(* CODESYS project Johnson,Joachim,Uppgift17_V2.project

Project tree, tasks and I/O mapping:
  Device : CODESYS Control Win V3, 3S - Smart Software Solutions GmbH, order no. 305021, version 3.5.10.40
    application Application
      libraries: Standard, * (System)
      task MainTask (cyclic, interval t#20ms, priority 1) calls PLC_PRG, Light [Handling Lights], ResetAlarm, PrintoutErrorMessages
      program PLC_PRG [LD]
      Symbols
      global variables GVL
      program Light [CFC]
      program ResetAlarm [CFC]
      program PrintoutErrorMessages [ST]
*)

// Device/Application/GVL
{attribute 'qualified_only'}
VAR_GLOBAL
		// signals from buttons
	iSUB00_S1: BOOL; // StartButton
	iSUB00_S2: BOOL; // Stopbutton
	iSUB00_S3: BOOL; // Resetbutton
	
	running: BOOL; 	 // Is the aplication running
	alarm: BOOL; 	 // Is the aplication running
	alarmcode: WORD; // handling the codes of the alarm
	
	Alarm1: BOOL;
	Alarm2: BOOL;
	Alarm3: BOOL;
	
	// Signals from conveyors
	iSUB01_B1: BOOL; // Signals för conveyor 1. ontop
	iSUB02_B1: BOOL; // Signals för conveyor 2. ontop
	iSUB03_B1: BOOL; // Signals för conveyor 3. ontop
	
	// Conveyor signal ontop conveyro
	oSUB00_H1: BOOL; // Auto-On light
	oSUB00_H2: BOOL; // Alarm light
	oSUB00_H3: WORD; // Display of errors
	oSUB01_K1: BOOL; // MOTOR FÖR converoyr 1
	oSUB02_K1: BOOL; // MOTOR FÖR converoyr 2
	oSUB03_K1: BOOL; // MOTOR FÖR converoyr 3
END_VAR

// Device/Application/PLC_PRG
PROGRAM PLC_PRG
VAR
	ReturnRunnongBool: BOOL;
	PressBtnTime: TIME;
	PressBtnTimer: TON;
	ONTOPCONRETURN: BOOL;
	ONTOPCONRETURN2: BOOL; // check that the previous con not take controll over engine/converour
	ONTOPCONRETURN3: BOOL; // check that the previous con not take controll over engine/converour
	TON_0: TON;
	TON_1: TON;
	TimElapseSincePastFirstSens: TIME;
	TON_2: TON;
	running: BOOL;
	ErrorCodePrintout: CTD;
	ErrorCodePrintout2: CTD;
	ErrorCodePrintout3: CTD;
	TimElapseSincePastFirstSens2: TIME;
	TON_3: TON;
	TON_4: TON;
	TimElapseSincePastFirstSens3: TIME;
	TimElapseSincePastFirstSens4: TIME;
	Alarm2: BOOL;
	Alarm1: BOOL;
	Alarm3: BOOL;
END_VAR
VAR // added by the converter: edge detectors and wires of the graphical bodies
    _w1, _w2, _w3, _w4, _w5, _w6 : BOOL;
END_VAR

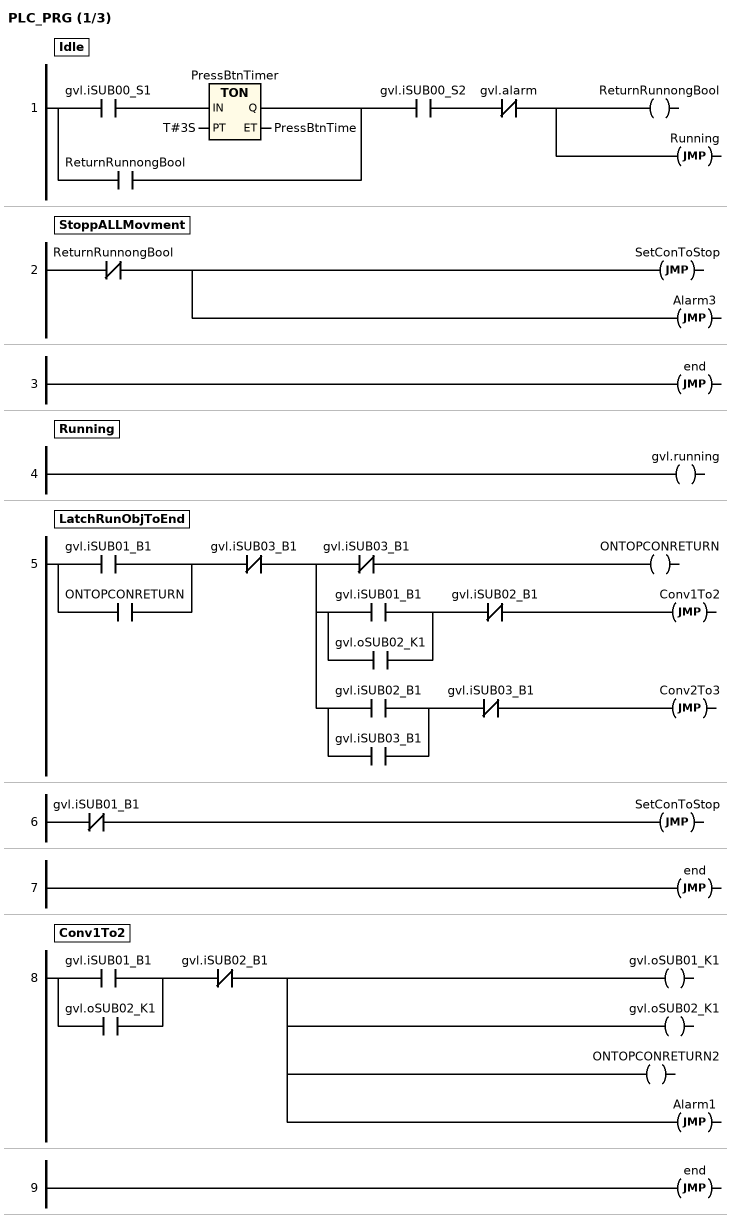
// NETWORK 1
Idle:
PressBtnTimer(IN := gvl.iSUB00_S1, PT := T#3S, ET => PressBtnTime); // TON
_w1 := ((PressBtnTimer.Q OR ReturnRunnongBool) AND gvl.iSUB00_S2) AND NOT gvl.alarm;
ReturnRunnongBool := _w1;
IF _w1 THEN JMP Running; END_IF

// NETWORK 2
StoppALLMovment:
_w2 := NOT ReturnRunnongBool;
IF _w2 THEN JMP SetConToStop; END_IF
IF _w2 THEN JMP Alarm3; END_IF

// NETWORK 3
JMP end;

// NETWORK 4
Running:
gvl.running := TRUE;

// NETWORK 5
LatchRunObjToEnd:
_w3 := (gvl.iSUB01_B1 OR ONTOPCONRETURN) AND NOT gvl.iSUB03_B1;
ONTOPCONRETURN := _w3 AND NOT gvl.iSUB03_B1;
IF (_w3 AND (gvl.iSUB01_B1 OR gvl.oSUB02_K1)) AND NOT gvl.iSUB02_B1 THEN JMP Conv1To2; END_IF
IF _w3 AND (gvl.iSUB02_B1 OR gvl.iSUB03_B1) AND NOT gvl.iSUB03_B1 THEN JMP Conv2To3; END_IF

// NETWORK 6
IF NOT gvl.iSUB01_B1 THEN JMP SetConToStop; END_IF

// NETWORK 7
JMP end;

// NETWORK 8
Conv1To2:
_w4 := (gvl.iSUB01_B1 OR gvl.oSUB02_K1) AND NOT gvl.iSUB02_B1;
gvl.oSUB01_K1 := _w4;
gvl.oSUB02_K1 := _w4;
ONTOPCONRETURN2 := _w4;
IF _w4 THEN JMP Alarm1; END_IF

// NETWORK 9
JMP end;

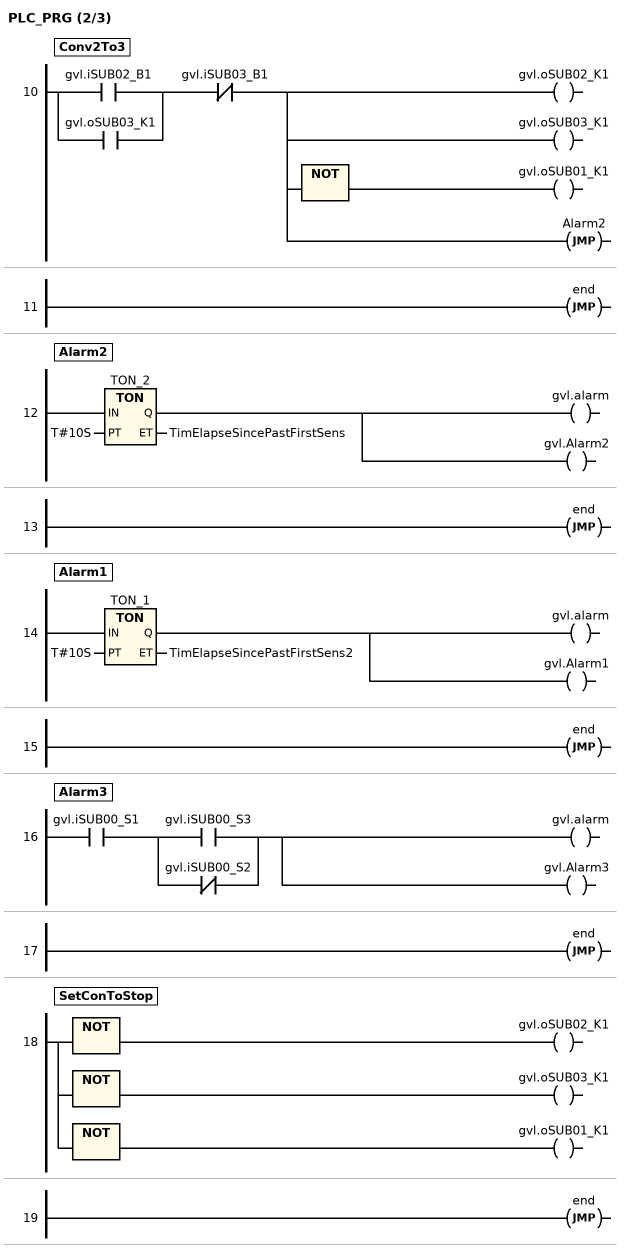
// NETWORK 10
Conv2To3:
_w5 := (gvl.iSUB02_B1 OR gvl.oSUB03_K1) AND NOT gvl.iSUB03_B1;
gvl.oSUB02_K1 := _w5;
gvl.oSUB03_K1 := _w5;
gvl.oSUB01_K1 := NOT _w5;
IF _w5 THEN JMP Alarm2; END_IF

// NETWORK 11
JMP end;

// NETWORK 12
Alarm2:
TON_2(IN := TRUE, PT := T#10S, ET => TimElapseSincePastFirstSens); // TON
gvl.alarm := TON_2.Q;
gvl.Alarm2 := TON_2.Q;

// NETWORK 13
JMP end;

// NETWORK 14
Alarm1:
TON_1(IN := TRUE, PT := T#10S, ET => TimElapseSincePastFirstSens2); // TON
gvl.alarm := TON_1.Q;
gvl.Alarm1 := TON_1.Q;

// NETWORK 15
JMP end;

// NETWORK 16
Alarm3:
_w6 := gvl.iSUB00_S1 AND (gvl.iSUB00_S3 OR NOT gvl.iSUB00_S2);
gvl.alarm := _w6;
gvl.Alarm3 := _w6;

// NETWORK 17
JMP end;

// NETWORK 18
SetConToStop:
gvl.oSUB02_K1 := NOT TRUE;
gvl.oSUB03_K1 := NOT TRUE;
gvl.oSUB01_K1 := NOT TRUE;

// NETWORK 19
JMP end;

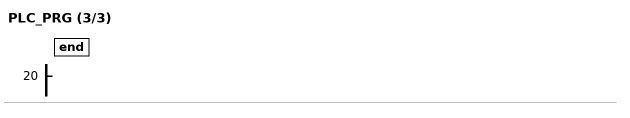
// NETWORK 20
end: ;

END_PROGRAM

// Device/Application/Light
PROGRAM Light
VAR
	Light_Time_TurnOff_Delayf: TON;
	TurnLightOffTimeoutpu: TIME;
	TurnLightOnTimeoutpu: TIME;
	Button_O: TON;
END_VAR
VAR // added by the converter: edge detectors and wires of the graphical bodies
    _w1 : BOOL;
END_VAR

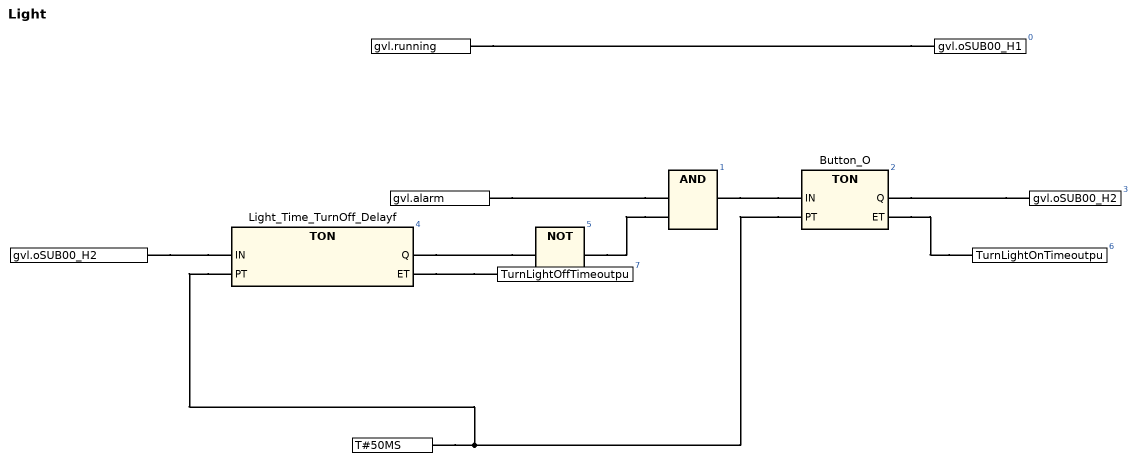
gvl.oSUB00_H1 := gvl.running;
Button_O(IN := gvl.alarm AND _w1, PT := T#50MS); // TON
gvl.oSUB00_H2 := Button_O.Q;
Light_Time_TurnOff_Delayf(IN := gvl.oSUB00_H2, PT := T#50MS); // TON
_w1 := NOT Light_Time_TurnOff_Delayf.Q;
TurnLightOnTimeoutpu := Button_O.ET;
TurnLightOffTimeoutpu := Light_Time_TurnOff_Delayf.ET;

END_PROGRAM

// Device/Application/ResetAlarm
PROGRAM ResetAlarm
VAR
END_VAR
VAR // added by the converter: edge detectors and wires of the graphical bodies
    _w1 : BOOL;
END_VAR

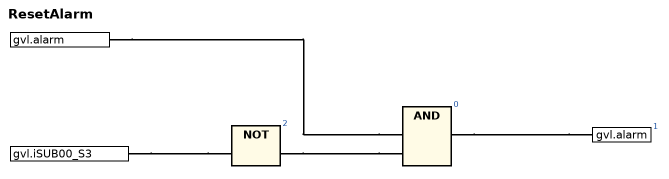
gvl.alarm := gvl.alarm AND _w1;
_w1 := NOT gvl.iSUB00_S3;

END_PROGRAM

// Device/Application/PrintoutErrorMessages
PROGRAM PrintoutErrorMessages
VAR
END_VAR

IF gvl.Alarm1 THEN
	gvl.oSUB00_H3 := 10;
END_IF

IF gvl.Alarm2 THEN
	gvl.oSUB00_H3 := 20;
END_IF

IF gvl.Alarm3 THEN
	gvl.oSUB00_H3 := 30;
END_IF

END_PROGRAM
